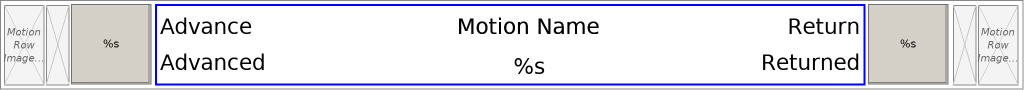
VISUALIZATION LanguageRow  // 1024x90
VAR_IN_OUT
	MotionRowInstanceSingle:typeMotionRow; //feedback to motion row to operator
	MotionRowButtonsSingle:typeMotionRowButtons; //button feedback in seperate interface
END_VAR
    Rectangle (155,4 710x81), invisible if: MotionRowInstanceSingle.Returned.bHideCoil AND MotionRowInstanceSingle.bHideName
    Button (868,4 80x80), "%s", text variable: MotionRowInstanceSingle.Returned.NumberOrder, invisible if: MotionRowInstanceSingle.Returned.bHideButton
        tap MotionRowButtonsSingle.btnReturn
    Button (71,4 80x80), "%s", text variable: MotionRowInstanceSingle.Advance.NumberOrder, invisible if: MotionRowInstanceSingle.Advance.bHideButton
        tap MotionRowButtonsSingle.btnAdvance
    Rectangle (393,50 273x33), "%s", text variable: MotionRowInstanceSingle.strPosn, invisible if: MotionRowInstanceSingle.bHidePosn
    Group (157,10 706x69)
        Rectangle (524,0 182x33), "Return", invisible if: MotionRowInstanceSingle.Returned.bHideCoil or MotionRowInstanceSingle.bIsAbsSymSwitch, text list: 'LanguageRowText', text index: MotionRowInstanceSingle.IndexLocation + 3, colour variable: MotionRowInstanceSingle.Returned.CoilColour
        Rectangle (235,0 273x33), "Motion Name", invisible if: MotionRowInstanceSingle.bHideName or MotionRowInstanceSingle.bIsAbsSymSwitch, text list: 'LanguageRowText', text index: MotionRowInstanceSingle.IndexLocation + 6
        Rectangle (524,36 182x33), "Returned", invisible if: MotionRowInstanceSingle.Returned.bHideDepth or MotionRowInstanceSingle.bIsAbsSymSwitch, text list: 'LanguageRowText', text index: MotionRowInstanceSingle.IndexLocation + 4, colour variable: MotionRowInstanceSingle.Returned.FdbkColour
        Rectangle (0,0 207x33), "Advance", text variable: MotionRowInstanceSingle.Advance.valCoil, invisible if: MotionRowInstanceSingle.Advance.bHideCoil or MotionRowInstanceSingle.bIsAbsSymSwitch, text list: 'LanguageRowText', text index: MotionRowInstanceSingle.IndexLocation + 0, colour variable: MotionRowInstanceSingle.Advance.CoilColour
        Rectangle (0,36 207x33), "Advanced", invisible if: MotionRowInstanceSingle.Advance.bHideDepth or MotionRowInstanceSingle.bIsAbsSymSwitch, text list: 'LanguageRowText', text index: MotionRowInstanceSingle.IndexLocation + 1, colour variable: MotionRowInstanceSingle.Advance.FdbkColour
    Image (4,5 40x80), invisible if: NOT MotionRowInstanceSingle.Advance.InterlockOK OR MotionRowInstanceSingle.Advance.bHideInterlock, image: MotionRowImages.LeftHighlight
    Image (4,5 40x80), invisible if: MotionRowInstanceSingle.Advance.InterlockOK OR MotionRowInstanceSingle.Advance.bHideInterlock, image: MotionRowImages.LeftNot
    Image (978,5 40x80), invisible if: MotionRowInstanceSingle.Returned.InterlockOK OR MotionRowInstanceSingle.Returned.bHideInterlock, image: MotionRowImages.RightNot
    Image (978,5 40x80), invisible if: NOT MotionRowInstanceSingle.Returned.InterlockOK OR MotionRowInstanceSingle.Returned.bHideInterlock, image: MotionRowImages.RightHighlight
    Image (46,5 23x80), invisible if: MotionRowInstanceSingle.Advance.Prompt OR MotionRowInstanceSingle.Advance.bHidePrompt, image: MotionRowImages.PromptNOK
    Image (953,5 23x80), invisible if: NOT MotionRowInstanceSingle.Returned.Prompt OR MotionRowInstanceSingle.Returned.bHidePrompt, image: MotionRowImages.PromptOK
    Image (953,5 23x80), invisible if: MotionRowInstanceSingle.Returned.Prompt OR MotionRowInstanceSingle.Returned.bHidePrompt, image: MotionRowImages.PromptNOK
    Image (46,5 23x80), invisible if: NOT MotionRowInstanceSingle.Advance.Prompt OR MotionRowInstanceSingle.Advance.bHidePrompt, image: MotionRowImages.PromptOK
    Group (157,10 706x69)
        Rectangle (524,0 182x33), "Return", invisible if: MotionRowInstanceSingle.Returned.bHideCoil or NOT MotionRowInstanceSingle.bIsAbsSymSwitch, text list: 'LanguageRowText', text index: MotionRowInstanceSingle.IndexLocation + 3 + 10, colour variable: MotionRowInstanceSingle.Returned.CoilColour
        Rectangle (235,0 273x33), "Motion Name", invisible if: MotionRowInstanceSingle.bHideName or NOT MotionRowInstanceSingle.bIsAbsSymSwitch, text list: 'LanguageRowText', text index: MotionRowInstanceSingle.IndexLocation + 6 + 10
        Rectangle (524,36 182x33), "Returned", invisible if: MotionRowInstanceSingle.Returned.bHideDepth or NOT MotionRowInstanceSingle.bIsAbsSymSwitch, text list: 'LanguageRowText', text index: MotionRowInstanceSingle.IndexLocation + 4 + 10, colour variable: MotionRowInstanceSingle.Returned.FdbkColour
        Rectangle (0,0 207x33), "Advance", text variable: MotionRowInstanceSingle.Advance.valCoil, invisible if: MotionRowInstanceSingle.Advance.bHideCoil or NOT MotionRowInstanceSingle.bIsAbsSymSwitch, text list: 'LanguageRowText', text index: MotionRowInstanceSingle.IndexLocation + 0 + 10, colour variable: MotionRowInstanceSingle.Advance.CoilColour
        Rectangle (0,36 207x33), "Advanced", invisible if: MotionRowInstanceSingle.Advance.bHideDepth or NOT MotionRowInstanceSingle.bIsAbsSymSwitch, text list: 'LanguageRowText', text index: MotionRowInstanceSingle.IndexLocation + 1 + 10, colour variable: MotionRowInstanceSingle.Advance.FdbkColour
END_VISUALIZATION

(* stored: Version 1.1.0.1, ProductVersion 3.1.4024.11
   Visu LanguageRow: Id {69dac12a-2317-0cdd-1cdd-77f7acb9b873} *)
